FUNCTION_BLOCK Time_Out_Actuator_CommandAndMoved (* Basic FB with empty ECC *)
  (* Standard: 61499-2 *)
  (* Version 1.0, 2023-03-16, AK125171 *)
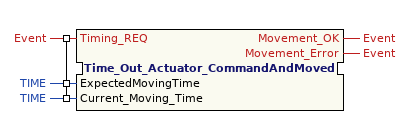
  EVENT_INPUT
    Timing_REQ WITH ExpectedMovingTime, Current_Moving_Time;
  END_EVENT
  EVENT_OUTPUT
    Movement_OK;
    Movement_Error;
  END_EVENT
  VAR_INPUT
    ExpectedMovingTime : TIME;
    Current_Moving_Time : TIME;
  END_VAR
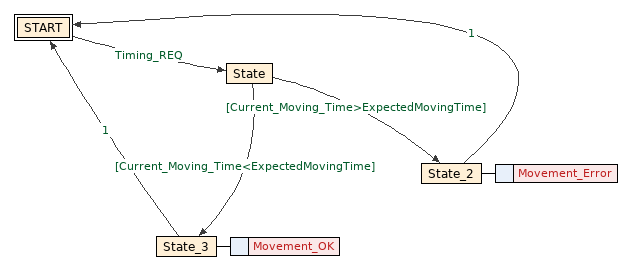
  EC_STATES
    START; (* Initial State *)
    State;
    State_2 : -> Movement_Error;
    State_3 : -> Movement_OK;
  END_STATES
  EC_TRANSITIONS
    START TO State := Timing_REQ;
    State TO State_3 := [Current_Moving_Time<ExpectedMovingTime];
    State TO State_2 := [Current_Moving_Time>ExpectedMovingTime];
    State_2 TO START := 1;
    State_3 TO START := 1;
  END_TRANSITIONS
END_FUNCTION_BLOCK
